{attribute 'qualified_only'}
{attribute 'strict'}
{attribute 'to_string'}
TYPE ST125_Cylinders_e :
(
    GreiferFilterhutLinks,
    GreiferFilterhutRechts,
    HandlingSolerohrLinks,
    HandlingSolerohrRechts,
    GreiferSolerohrLinks,
    GreiferSolerohrRechts,
    _max
);
END_TYPE

(* stored: Version 1.1.0.1, ProductVersion 3.1.4024.6
   EnumerationTextList ST125_Cylinders_e: Id {c7aab1ff-26dc-4777-9069-6a1c1f601c61} *)
